INTERFACE I_Brake

END_INTERFACE

(* stored: Version 1.1.0.1
   Itf I_Brake: Id {190f63fb-756a-4791-8091-567b83a9d052} *)
